# EPICS autosave request: IOCs/12id/iocBoot/ioc12idb/asynRecord.req
$(P).SCAN
$(P).TMOD
$(P).OEOS
$(P).IEOS
$(P).OFMT
$(P).IFMT
$(P).TMOT
$(P).NRRD
$(P).BAUD
$(P).DBIT
$(P).SBIT
$(P).PRTY
$(P).MCTL
$(P).FCTL
$(P).DESC
